Omron CX-Programmer project NewProject (CX-Programmer 9.51)

# PLC My_First_Project: CP1L L
; MyFirstProject

## Global symbols (name address type ; comment)
150 CHANNEL  ; Timer number
T0002 BOOL  ; Timer number
T0003 BOOL  ; Timer number

## Program NewProgram1 (cyclic task 0)
Local symbols
button_2 0.01 BOOL
out_3 100.02 BOOL

### Section Section1

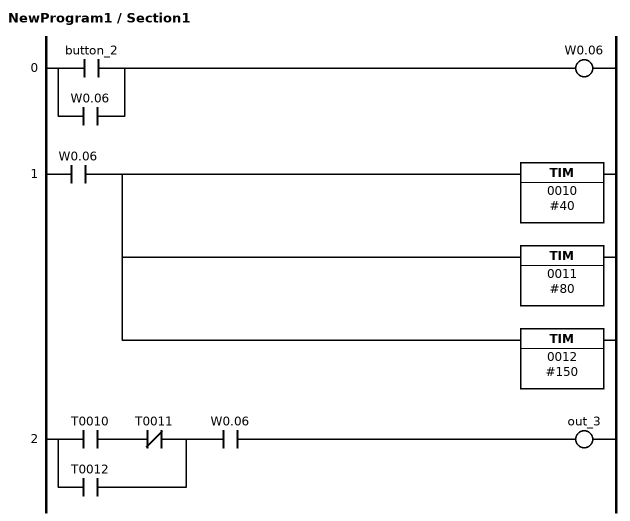
; rung 0
LD button_2
OR W0.06
OUT W0.06
; rung 1
LD W0.06
TIM 0010 #40
TIM 0011 #80
TIM 0012 #150
; rung 2
LD T0010
ANDNOT T0011
OR T0012
AND W0.06
OUT out_3

### Section END
; rung 0
END(001)